PROGRAM MAIN
VAR
	traError			: BOOL;
	traInitDone			: BOOL;
	bModeOff			: BOOL;
	bModeManual			: BOOL := TRUE;
	bModeAuto			: BOOL;
	Err_T				: R_TRIG;
	Wrn_T				: R_TRIG;
	Wrn_T1				: R_TRIG;
	Reset_T				: R_TRIG;
	fbtimer				: TON;
	fbTimerSirens		: TON;
	fbTimer_IoT			: Ton;
	Run_T				: R_TRIG;
	Stop_T				: R_TRIG;
	k,k1				: INT;
	nState				: INT;
	nStateEmr			: INT;
	nState2				: INT;
	nState_IoT			: INT;
	bFaultFlag			: BOOL;
	nstateStop			: INT;
	fbTimerStop			: TON;
	timerStop			: ton;
	timerReset			: TON;
	nWriteData			: INT;
	TimerData			: TON;
	FbTimerModbus		: ARRAY [1..7] OF TON;
	fbEventlogger		: FB_Eventlogger;
	fbEventButton		: FB_EventButton;
	nstatechange		: INT;
	bWriteAlarm			: BOOL;
END_VAR

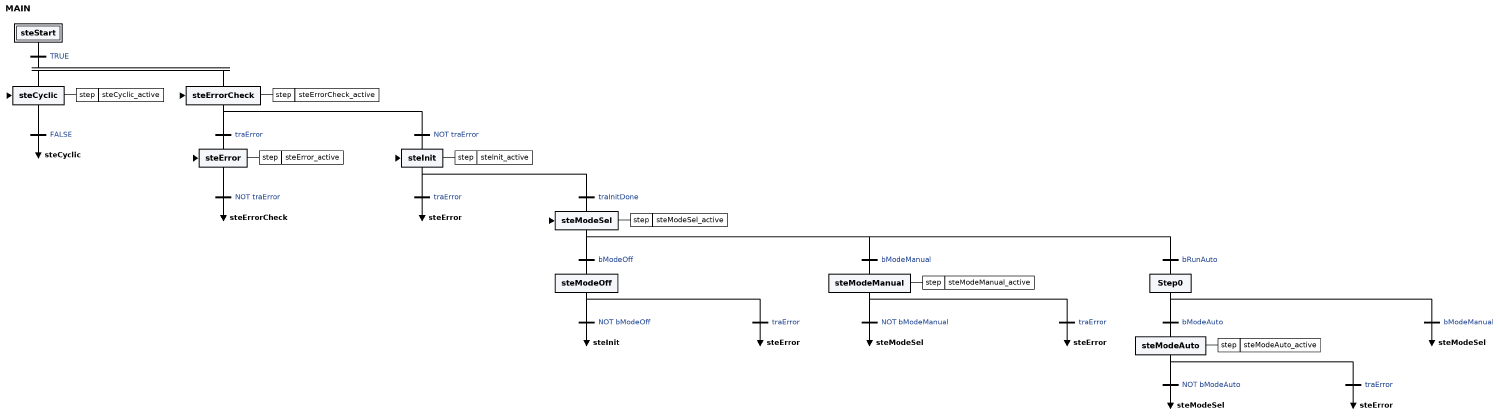
INITIAL_STEP steStart:
END_STEP
TRANSITION FROM steStart TO (steCyclic, steErrorCheck)
    := TRUE;
END_TRANSITION
STEP steCyclic:
    steCyclic_active(N);  // step action
END_STEP
TRANSITION FROM steCyclic TO steCyclic
    := FALSE;
END_TRANSITION
STEP steErrorCheck:
    steErrorCheck_active(N);  // step action
END_STEP
TRANSITION FROM steErrorCheck TO steError
    := traError;
END_TRANSITION
STEP steError:
    steError_active(N);  // step action
END_STEP
TRANSITION FROM steError TO steErrorCheck
    := NOT traError;
END_TRANSITION
TRANSITION FROM steErrorCheck TO steInit
    := NOT traError;
END_TRANSITION
STEP steInit:
    steInit_active(N);  // step action
END_STEP
TRANSITION FROM steInit TO steError
    := traError;
END_TRANSITION
TRANSITION FROM steInit TO steModeSel
    := traInitDone;
END_TRANSITION
STEP steModeSel:
    steModeSel_active(N);  // step action
END_STEP
TRANSITION FROM steModeSel TO steModeOff
    := bModeOff;
END_TRANSITION
STEP steModeOff:
END_STEP
TRANSITION FROM steModeOff TO steInit
    := NOT bModeOff;
END_TRANSITION
TRANSITION FROM steModeOff TO steError
    := traError;
END_TRANSITION
TRANSITION FROM steModeSel TO steModeManual
    := bModeManual;
END_TRANSITION
STEP steModeManual:
    steModeManual_active(N);  // step action
END_STEP
TRANSITION FROM steModeManual TO steModeSel
    := NOT bModeManual;
END_TRANSITION
TRANSITION FROM steModeManual TO steError
    := traError;
END_TRANSITION
TRANSITION FROM steModeSel TO Step0
    := bRunAuto;
END_TRANSITION
STEP Step0:
END_STEP
TRANSITION FROM Step0 TO steModeAuto
    := bModeAuto;
END_TRANSITION
TRANSITION FROM Step0 TO steModeSel
    := bModeManual;
END_TRANSITION
STEP steModeAuto:
    steModeAuto_active(N);  // step action
END_STEP
TRANSITION FROM steModeAuto TO steModeSel
    := NOT bModeAuto;
END_TRANSITION
TRANSITION FROM steModeAuto TO steError
    := traError;
END_TRANSITION

ACTION ListError:
Err_T(CLK := bError1);
Wrn_T(CLK := bWarning);

IF i > 100 THEN
	i := 100;
END_IF
		
CASE nState OF 
	0:
		IF Err_T.Q THEN
			nState := 1;
		ELSIF Wrn_T.Q THEN
			bWrn := TRUE;
			nState := 10;
		END_IF

	1:
		CASE nErrorID OF
			1:
				stErrorTxt := "E1_1.Lỗi hết hũ trạm 1 [kiểm tra U1I5-2]";
				stErrorTxt1 := 'E1_1.The jar is empty line 1 [check U1I5-2]';
				fbEventlogger(eventClass := TC_EVENTS.Entobel.Event1.uuidEventClass, nEventID := DINT_TO_UDINT(nErrorID));
			2:
				stErrorTxt := "E2_1.Lỗi hũ bị kẹt trạm 1 [kiểm tra U1I5-6]";
				stErrorTxt1 := 'E2_1.The jar  is trapped line 1 [check U1I5-6]';
				fbEventlogger(eventClass := TC_EVENTS.Entobel.Event2.uuidEventClass, nEventID := DINT_TO_UDINT(nErrorID));
			3:
				stErrorTxt := "E3_1.Lỗi ben chặn hũ trên rút về trạm 1 [kiểm tra U1I5-3]" ;
				stErrorTxt1 := 'E3_1.The upper cylinder retract  is faulty line 1 [check U1I5-3]';
				fbEventlogger(eventClass := TC_EVENTS.Entobel.Event3.uuidEventClass, nEventID := DINT_TO_UDINT(nErrorID));
			4:
				stErrorTxt := "E4_1.Lỗi ben chặn hũ dưới rút về trạm 1 [kiểm tra U1I5-4]";
				stErrorTxt1 := 'E4_1.The lower cylinder retract  is faulty line 1 [check U1I5-4]';
				fbEventlogger(eventClass := TC_EVENTS.Entobel.Event4.uuidEventClass, nEventID := DINT_TO_UDINT(nErrorID));
			5:
				stErrorTxt := "E5_1.Lỗi ben chặn hũ dưới đẩy ra trạm 1 [kiểmtra U1I5-5]";
				stErrorTxt1 := 'E5_1.The lower cylinder extend  is faulty line 1 [check U1I5-5]';
				fbEventlogger(eventClass := TC_EVENTS.Entobel.Event5.uuidEventClass, nEventID := DINT_TO_UDINT(nErrorID));
			6:
				stErrorTxt := "E6_1.Lỗi biến tần đảo thức ăn trạm 1 [kiểm tra biến tần 4]";
				stErrorTxt1 := 'E6_1.The inverter of agitator motor fault line 1 [check U1I5-6]';
				fbEventlogger(eventClass := TC_EVENTS.Entobel.Event6.uuidEventClass, nEventID := DINT_TO_UDINT(nErrorID));
			7:
				stErrorTxt := "E7_1.Lỗi driver chia thức ăn trạm 1 [kiểm tra driver 2]";
				stErrorTxt1 := 'E7_1.The driver of dispenser motor fault line 1 [check driver 2]';
				fbEventlogger(eventClass := TC_EVENTS.Entobel.Event7.uuidEventClass, nEventID := DINT_TO_UDINT(nErrorID));
			8:
				stErrorTxt := "E8_1.Lỗi ben chặn sâu rút về trạm 1 [kiểm tra U1I5-7]";
				stErrorTxt1 := 'E8_1.The cylinder blocking worm retract  is faulty line 1 [check U1I5-7]';
				fbEventlogger(eventClass := TC_EVENTS.Entobel.Event8.uuidEventClass, nEventID := DINT_TO_UDINT(nErrorID));
			9:
				stErrorTxt := "E9_1.Lỗi biến tần phểu rung sâu trạm 1 [kiểm tra biến tần 5]";
				stErrorTxt1 := 'E9_1.The inverter of vibrating funnel fault line 1 [check inverter 5]';
				fbEventlogger(eventClass := TC_EVENTS.Entobel.Event9.uuidEventClass, nEventID := DINT_TO_UDINT(nErrorID));
			10:
				stErrorTxt := "E10_1.Lỗi hết nắp trạm 1 [kiểm tra U1I5-8]";
				stErrorTxt1 := 'E10_1.The lid is empty line 1 [check U1I5-8]';
				fbEventlogger(eventClass := TC_EVENTS.Entobel.Event10.uuidEventClass, nEventID := DINT_TO_UDINT(nErrorID));
			11:
				stErrorTxt := "E11_1.Lỗi ben chặn nắp rút về trạm 1 [kiểm tra U1I6-1]";
				stErrorTxt1 := 'E11_1.The cylinder blocking the lid retract is faulty line 1 [check U1I6-1]';
				fbEventlogger(eventClass := TC_EVENTS.Entobel.Event11.uuidEventClass, nEventID := DINT_TO_UDINT(nErrorID));
			12:
				stErrorTxt := "E12-1.Lỗi ben chặn nắp đẩy ra trạm 1 [kiểm tra U1I6-2]";
				stErrorTxt1 := 'E12_1.The cylinder blocking the lid extend is faulty line 1 [check U1I6-2]';
				fbEventlogger(eventClass := TC_EVENTS.Entobel.Event12.uuidEventClass, nEventID := DINT_TO_UDINT(nErrorID));
			13:
				stErrorTxt := "E13_1.Lỗi ben hút/thả nắp rút về trạm 1 [kiểm tra U1I6-3]";
				stErrorTxt1 := 'E13_1.The cylinder sucking the lid retract is faulty line 1 [check U1I6-3]';
				fbEventlogger(eventClass := TC_EVENTS.Entobel.Event13.uuidEventClass, nEventID := DINT_TO_UDINT(nErrorID));
			14:
				stErrorTxt := "E14_1.Lỗi ben hút/thả nắp đẩy ra trạm 1 [kiểm tra U1I6-4]";
				stErrorTxt1 := 'E14_1.The cylinder sucking the lid extend is faulty line 1 [check U1I6-4]';
				fbEventlogger(eventClass := TC_EVENTS.Entobel.Event14.uuidEventClass, nEventID := DINT_TO_UDINT(nErrorID));
			15:
				stErrorTxt := "E15_1.Lỗi ben dập nắp rút về trạm 1 [kiểm tra U1I6-6]";
				stErrorTxt1 := 'E15_1.The cylinder pressing the lid retract is faulty line 1 [check U1I6-6]';
				fbEventlogger(eventClass := TC_EVENTS.Entobel.Event15.uuidEventClass, nEventID := DINT_TO_UDINT(nErrorID));
			16:
				stErrorTxt := "E16_1.Lỗi ben dập nắp đẩy ra trạm 1 [kiểm tra U1I6-7]";
				stErrorTxt1 := 'E16_1.The cylinder pressing the lid extend is faulty line 1 [check U1I6-7]';
				fbEventlogger(eventClass := TC_EVENTS.Entobel.Event16.uuidEventClass, nEventID := DINT_TO_UDINT(nErrorID));
			17:
				stErrorTxt := "E17_1.Lỗi ben lượt ra/vào rút về trạm 1 [kiểm tra U1I6-8]";
				stErrorTxt1 := 'E17_1.The comb cylinder retract is faulty line 1 [check U1I6-8]';
				fbEventlogger(eventClass := TC_EVENTS.Entobel.Event17.uuidEventClass, nEventID := DINT_TO_UDINT(nErrorID));
			18:
				stErrorTxt := "E18_1.Lỗi ben lượt ra/vào đẩy ra trạm 1 [kiểm tra U1I7-1]";
				stErrorTxt1 := 'E18_1.The comb cylinder extend is faulty line 1 [check U1I7-1]';
				fbEventlogger(eventClass := TC_EVENTS.Entobel.Event18.uuidEventClass, nEventID := DINT_TO_UDINT(nErrorID));
			19:
				stErrorTxt := "E19_1.Lỗi ben kẹp hũ rút về trạm 1 [kiểm tra U1I7-4]";
				stErrorTxt1 := 'E19_1.The clap cylinder retract is faulty line 1 [check U1I7-4]';
				fbEventlogger(eventClass := TC_EVENTS.Entobel.Event19.uuidEventClass, nEventID := DINT_TO_UDINT(nErrorID));
			20:
				stErrorTxt := "E20_1.Lỗi ben kẹp hũ đẩy ra trạm 1 [kiểm tra U1I7-5]";	
				stErrorTxt1 := 'E20_1.The clap cylinder extend is faulty line 1 [check U1I7-5]';
				fbEventlogger(eventClass := TC_EVENTS.Entobel.Event20.uuidEventClass, nEventID := DINT_TO_UDINT(nErrorID));
			21:
				stErrorTxt := "E21_1.Lỗi ben di chuyển lượt rút về trạm 1 [kiểm tra U1I7-2]";	
				stErrorTxt1 := 'E21_1.The cylinder moving comb retract is faulty line 1 [check U1I7-2]';
				fbEventlogger(eventClass := TC_EVENTS.Entobel.Event21.uuidEventClass, nEventID := DINT_TO_UDINT(nErrorID));
			22:
				stErrorTxt := "E22_1.Lỗi ben di chuyển lượt đẩy ra trạm 1 [kiểm tra U1I7-3]";
				stErrorTxt1 := 'E22_1.The cylinder moving comb extend is faulty line 1 [check U1I7-3]';
				fbEventlogger(eventClass := TC_EVENTS.Entobel.Event22.uuidEventClass, nEventID := DINT_TO_UDINT(nErrorID));
			45:
				stErrorTxt := "E23_1.Lỗi mất hũ khi đang cân thức ăn trạm 1 [kiểm tra U1I7-6]";
				stErrorTxt1 := 'E23_1.The jar is missed when weighting food line 1 [check U1I7-6]';
				fbEventlogger(eventClass := TC_EVENTS.Entobel.Event45.uuidEventClass, nEventID := DINT_TO_UDINT(nErrorID));
			47:
				stErrorTxt := "E24_1.Lỗi mất hũ khi đang cân sâu trạm 1 [kiểm tra U1I7-7]";
				stErrorTxt1 := 'E24_1.The jar is missed when weighting larvae line 1 [check U1I7-7]';
				fbEventlogger(eventClass := TC_EVENTS.Entobel.Event47.uuidEventClass, nEventID := DINT_TO_UDINT(nErrorID));
			49:
				stErrorTxt := "E25_1.Lỗi hút không được nắp trạm 1 [kiểm tra U1I6-5]";
				stErrorTxt1 := 'E25_1.Failed to suction the lid line 1 [check U1I6-5]';
				fbEventlogger(eventClass := TC_EVENTS.Entobel.Event49.uuidEventClass, nEventID := DINT_TO_UDINT(nErrorID));
			51:
				stErrorTxt := "E26_1.Lỗi nắp đã được hút trạm 1 [kiểm tra U1I6-5]";
				stErrorTxt1 := 'E26_1.The lid is still on the valve line 1 [check U1I5-6]';	
				fbEventlogger(eventClass := TC_EVENTS.Entobel.Event51.uuidEventClass, nEventID := DINT_TO_UDINT(nErrorID));
			53:
				stErrorTxt := "E27_1.Lỗi an toàn cửa 1 [kiểm tra U1I7-8]";	
				stErrorTxt1 := 'E27_1.The safety door 1 is error [check U1I7-8]';	
				fbEventlogger(eventClass := TC_EVENTS.Entobel.Event53.uuidEventClass, nEventID := DINT_TO_UDINT(nErrorID));
			54:
				stErrorTxt := "E28_1.Lỗi an toàn cửa 2 [kiểm tra U1I7-9]";
				stErrorTxt1 := 'E28_1.The safety door 2 is error [check U1I7-9]';	
				fbEventlogger(eventClass := TC_EVENTS.Entobel.Event54.uuidEventClass, nEventID := DINT_TO_UDINT(nErrorID));
			55:
				stErrorTxt := "E29_1.Lỗi an toàn cửa 3 [kiểm tra U1I7-10]";
				stErrorTxt1 := 'E29_1.The safety door 3 is error [check U1I7-10]';
				fbEventlogger(eventClass := TC_EVENTS.Entobel.Event55.uuidEventClass, nEventID := DINT_TO_UDINT(nErrorID));	
			56: 
				stErrorTxt := "E30_1.Lỗi quá cân thức ăn trạm 1 [kiểm tra cân thức ăn]";
				stErrorTxt1 := 'E30_1.Overload weightfood [check U1I5-6]';	
				fbEventlogger(eventClass := TC_EVENTS.Entobel.Event56.uuidEventClass, nEventID := DINT_TO_UDINT(nErrorID));
			57: 
				stErrorTxt := "E31_1.Lỗi quá cân sâu trạm 1 [kiểm tra cân sâu]";
				stErrorTxt1 := 'E30_1.Overload weightLarvae [check U1I5-6]';
				fbEventlogger(eventClass := TC_EVENTS.Entobel.Event57.uuidEventClass, nEventID := DINT_TO_UDINT(nErrorID));	
			60:
				stErrorTxt := "E32_1.Lỗi ben hút/thả hũ đẩy ra trạm 1 [kiểm tra U1I7-11]";
				stErrorTxt1 := 'E32_1.The cylinder sucking the jar is faulty line 1 [check U1I7-11]';
				fbEventlogger(eventClass := TC_EVENTS.Entobel.Event60.uuidEventClass, nEventID := DINT_TO_UDINT(nErrorID)); 
			64:
				stErrorTxt := "E33_1.Lỗi Modbus thiết bị 3";
				stErrorTxt1 := 'E33_1.Error Modbus device 3';
				fbEventlogger(eventClass := TC_EVENTS.Entobel.Event64.uuidEventClass, nEventID := DINT_TO_UDINT(nErrorID));	
			65:
				stErrorTxt := "E34_1.Lỗi Modbus thiết bị 4";
				stErrorTxt1 := 'E34_1.Error Modbus device 4';
				fbEventlogger(eventClass := TC_EVENTS.Entobel.Event65.uuidEventClass, nEventID := DINT_TO_UDINT(nErrorID));	
			66:
				stErrorTxt := "E35_1.Lỗi Modbus thiết bị 5";
				stErrorTxt1 := 'E35_1.Error Modbus device 5';
				fbEventlogger(eventClass := TC_EVENTS.Entobel.Event66.uuidEventClass, nEventID := DINT_TO_UDINT(nErrorID));	
			68:
				stErrorTxt := "E36_1.Lỗi Modbus thiết bị 7";
				stErrorTxt1 := 'E36_1.Error Modbus device 7';
				fbEventlogger(eventClass := TC_EVENTS.Entobel.Event68.uuidEventClass, nEventID := DINT_TO_UDINT(nErrorID));	
			69:
				stErrorTxt := "E37_1.Lỗi đầu cân thức ăn Mettler Toledo 1";
				stErrorTxt1 := 'E37_1.Error Mettler Toledo 1';
				fbEventlogger(eventClass := TC_EVENTS.Entobel.Event69.uuidEventClass, nEventID := DINT_TO_UDINT(nErrorID));	
			70:
				stErrorTxt := "E38_1.Lỗi đầu cân sâu Mettler Toledo 2";
				stErrorTxt1 := 'E38_1.Error Mettler Toledo 2';
				fbEventlogger(eventClass := TC_EVENTS.Entobel.Event70.uuidEventClass, nEventID := DINT_TO_UDINT(nErrorID));	
			73:
				stErrorTxt := "E39_1.Lỗi ben chặn sâu đẩy ra trạm 1 [kiểm tra U1I5-7]";
				stErrorTxt1 := 'E39_1.The cylinder blocking worm extend  is faulty line 1';
				fbEventlogger(eventClass := TC_EVENTS.Entobel.Event73.uuidEventClass, nEventID := DINT_TO_UDINT(nErrorID));	
			75:
				stErrorTxt := "E40_1.Lỗi thiếu khí đầu vào [kiểm tra U1I7-13]";
				stErrorTxt1 := 'E40_1.Error of lack of input air [check U1I7-13]';
				fbEventlogger(eventClass := TC_EVENTS.Entobel.Event75.uuidEventClass, nEventID := DINT_TO_UDINT(nErrorID));	
			76:
				stErrorTxt := "E41_1.Lỗi hết thức ăn trạm 1";
				stErrorTxt1 := 'E41_1.Error running out of food line 1';
				fbEventlogger(eventClass := TC_EVENTS.Entobel.Event76.uuidEventClass, nEventID := DINT_TO_UDINT(nErrorID));	
			77:
				stErrorTxt := "E42_1.Lỗi hết sâu trạm 1";
				stErrorTxt1 := 'E42_1.Error running out of larvae line 1';
				fbEventlogger(eventClass := TC_EVENTS.Entobel.Event78.uuidEventClass, nEventID := DINT_TO_UDINT(nErrorID));		
			98:
				stErrorTxt := "E98_1.Dừng khẩn [kiểm tra Emergency]";
				stErrorTxt1 := 'E98_1.Emergency Stop [check Emergency]';
				fbEventlogger(eventClass := TC_EVENTS.Entobel.Event98.uuidEventClass, nEventID := DINT_TO_UDINT(nErrorID));	 
			99: 
				stErrorTxt := "E99_1.Lỗi biến tần băng tải đầu ra [kiểm tra biến tần 3]";
				stErrorTxt1 := 'E99_1.The inverter of conveyor out [check inverter 3]';	
				fbEventlogger(eventClass := TC_EVENTS.Entobel.Event99.uuidEventClass, nEventID := DINT_TO_UDINT(nErrorID));
		END_CASE
		IF i <> 1 THEN
			FOR	k := i TO 2 BY -1 DO
				nErrorIDList1[k].nErrorID 	 := nErrorIDList1[k-1].nErrorID;
				nErrorIDList1[k].ErrorTime   := nErrorIDList1[k-1].ErrorTime;
				nErrorIDList1[k].ErrorStatus := nErrorIDList1[k-1].ErrorStatus;	
			END_FOR		
		END_IF 
		nErrorIDList1[1].nErrorID := nErrorID;
		nErrorIDList1[1].ErrorTime := SYSTEMTIME_TO_DT(GetLocalSystemTime.systemTime);
		nErrorIDList1[1].ErrorStatus := 1;
		nStatus1	:= 'ERROR';
		i := i + 1;
		bWarning := FALSE;
		bTo_alarm_side := TRUE;
		nState := 2;
	2:
		bWriteAlarm	:= TRUE;
		bSirens := TRUE;
		nState := 3;
	3:
		IF NOT bError1 THEN
			nState 	:= 0;
			bSirens := FALSE;
		END_IF
	10:
		CASE nWarningID OF
			101:
				stWarningTxt := "W1_1.Cảnh báo hết hũ trạm 1[kiểm tra U1I5-2]";
				stWarningTxt1 := 'W1_1.Warning out of jar line 1 [check U1I5-2]';
				fbEventlogger(eventClass := TC_EVENTS.Entobel.Event101.uuidEventClass, nEventID := DINT_TO_UDINT(nWarningID));
			102:
				stWarningTxt := "W2_1.Cảnh báo hết nắp trạm 1[kiểm tra U1I5-8]";
				stWarningTxt1 := 'W2_1.Warning out of lid line 1 [check U1I5-8]';
				fbEventlogger(eventClass := TC_EVENTS.Entobel.Event102.uuidEventClass, nEventID := DINT_TO_UDINT(nWarningID));
			103:
				stWarningTxt := "W3_1.Cảnh báo hết thức ăn trạm 1";
				stWarningTxt1 := 'W3_1.Warning running out of food line 1';
				fbEventlogger(eventClass := TC_EVENTS.Entobel.Event103.uuidEventClass, nEventID := DINT_TO_UDINT(nWarningID));
			104:
				stWarningTxt := "W4_1.Cảnh báo cân quá khối lượng thức ăn trạm 1";
				stWarningTxt1 := 'W4_1.Warning food weight exceeds limit line 1';
				fbEventlogger(eventClass := TC_EVENTS.Entobel.Event104.uuidEventClass, nEventID := DINT_TO_UDINT(nWarningID));
			105:
				stWarningTxt := "W5_1.Cảnh báo hết sâu trạm 1";
				stWarningTxt1 := 'W5_1.Warning running out of larvae line 1';
				fbEventlogger(eventClass := TC_EVENTS.Entobel.Event105.uuidEventClass, nEventID := DINT_TO_UDINT(nWarningID));
			106:
				stWarningTxt := "W6_1.Canh bao can qua khoi luong sau tram 1";
				stWarningTxt1 := 'W6_1.Warning larvae weight exceeds limit line 1';
				fbEventlogger(eventClass := TC_EVENTS.Entobel.Event106.uuidEventClass, nEventID := DINT_TO_UDINT(nWarningID));
			107:
				stWarningTxt := "W7_1.Cảnh báo dập nắp không vô trạm 1[kiểm tra U1I6-7]";
				stWarningTxt1 := 'W7_1.Warning do not press lid inward line 1 [check U1I6-7]';
				fbEventlogger(eventClass := TC_EVENTS.Entobel.Event107.uuidEventClass, nEventID := DINT_TO_UDINT(nWarningID));
			115:
				stWarningTxt := "W8_1.Cảnh báo mất kết nối với PC Advantech [kiểm tra PC]";
				stWarningTxt1 := 'W8_1.Warning disconnect to PC Advantech [check PC]';	
				bAlarm_Iot := TRUE;	
		END_CASE
		IF i <> 1 THEN
			FOR	k := i TO 2 BY -1 DO
				nErrorIDList1[k].nErrorID 	 := nErrorIDList1[k-1].nErrorID;
				nErrorIDList1[k].ErrorTime   := nErrorIDList1[k-1].ErrorTime;
				nErrorIDList1[k].ErrorStatus := nErrorIDList1[k-1].ErrorStatus;		
			END_FOR		
		END_IF 
		nErrorIDList1[1].nErrorID := nWarningID;
		nErrorIDList1[1].ErrorTime := SYSTEMTIME_TO_DT(GetLocalSystemTime.systemTime);
		nErrorIDList1[1].ErrorStatus := 1;
		nStatus1	:= 'WARNING';
		i := i + 1;
		nState := 11;
	11:
		bWriteAlarm	:= TRUE;
		bSirens := TRUE;
		nState := 12;
	12:
		bWarning := FALSE;
		nState := 0;		
END_CASE

IF bclearall THEN
	FOR k := 1 TO 100 DO
		AlarmList[1,k] := "";
		AlarmList[2,k] := "";	
		AlarmList[3,k] := "";
		AlarmList[4,k] := "";	
		AlarmList3[1,k] := '';
		AlarmList3[2,k] := '';	
		AlarmList3[3,k] := '';
		AlarmList3[4,k] := '';	
	END_FOR
	i := 1;
END_IF

IF username <> '' THEN
	IF getuser = 'Operator' THEN
		IF NOT bSafetyDoor1 THEN
			F_SetError(53,nLine := 3);
		ELSIF NOT bSafetyDoor2 THEN
			F_SetError(54,nLine := 3);	
		ELSIF NOT bSafetyDoor3 THEN
			F_SetError(55,nLine := 3);	
		END_IF
		bypass := FALSE;
		hienthibypass := FALSE;
	ELSIF getuser = 'Engineer' THEN
		hienthibypass := TRUE;
		IF NOT bypass THEN
			IF NOT bSafetyDoor1 THEN
				F_SetError(53,nLine := 3);
			ELSIF NOT bSafetyDoor2 THEN
				F_SetError(54,nLine := 3);	
			ELSIF NOT bSafetyDoor3 THEN
				F_SetError(55,nLine := 3);	
			END_IF
		END_IF
	END_IF
END_IF
IF username <> '' THEN
	IF Error[1] THEN 
		(*IF ErrorID[1] = 150 OR ErrorID[1] = 32 THEN
			FbTimerModbus[1](IN := FALSE, PT := T#1S);
		ELSE*)
			//FbTimerModbus[1](IN := TRUE, PT := T#1S);
			//IF FbTimerModbus[1].Q  THEN
				F_SetError(62,nLine := 2);
			//END_IF
		//END_IF
	ELSE
		FbTimerModbus[1](IN := FALSE);
	END_IF
	
	IF Error[2] THEN
		(*IF ErrorID[2] = 150 OR ErrorID[2] = 32 THEN
			FbTimerModbus[2](IN := FALSE, PT := T#1S);
		ELSE*)
			//FbTimerModbus[2](IN := TRUE, PT := T#1S);
			//IF FbTimerModbus[2].Q THEN
				F_SetError(63,nLine := 2);
			//END_IF
		//END_IF
	ELSE
		FbTimerModbus[2](IN := FALSE);
	END_IF
	
	IF Error[3] THEN
		(*IF ErrorID[3] = 150 OR ErrorID[3] = 32 THEN
			FbTimerModbus[3](IN := FALSE, PT := T#1S);
		ELSE*)
			//FbTimerModbus[3](IN := TRUE, PT := T#1S);
			//IF FbTimerModbus[3].Q THEN
				F_SetError(64,nLine := 3);
				PR_Conveyor_Out.Stop();
				bRun := FALSE;
			//END_IF
		//END_IF
	ELSE
		FbTimerModbus[3](IN := FALSE);
	END_IF
	
	IF Error[4] THEN
		(*IF ErrorID[4] = 150 OR ErrorID[4] = 32 THEN
			FbTimerModbus[4](IN := FALSE, PT := T#1S);
		ELSE *)
			//FbTimerModbus[4](IN := TRUE, PT := T#1S);
			//IF FbTimerModbus[4].Q THEN
				F_SetError(65,nLine := 1);
			//END_IF
		//END_IF
	ELSE
		FbTimerModbus[4](IN := FALSE);
	END_IF
	
	IF Error[5] THEN
		(*IF ErrorID[5] = 150 OR ErrorID[5] = 32 THEN
			FbTimerModbus[5](IN := FALSE, PT := T#1S);
		ELSE*)
			//FbTimerModbus[5](IN := TRUE, PT := T#1S);
			//IF FbTimerModbus[5].Q THEN
				F_SetError(66,nLine := 1);
			//END_IF
		//END_IF
	ELSE
		FbTimerModbus[5](IN := FALSE);
	END_IF
	
	IF Error[6] THEN
		(*IF ErrorID[6] = 150 OR ErrorID[6] = 32 THEN
			FbTimerModbus[6](IN := FALSE, PT := T#1S);
		ELSE*)
			//FbTimerModbus[6](IN := TRUE, PT := T#1S);
			//IF FbTimerModbus[6].Q THEN
				F_SetError(67,nLine := 2);
			//END_IF
		//END_IF
	ELSE
		FbTimerModbus[6](IN := FALSE);
	END_IF
	
	IF Error[7] THEN
		(*IF ErrorID[2] = 150 OR ErrorID[7] = 32 THEN
			FbTimerModbus[7](IN := FALSE, PT := T#1S);
		ELSE*)
			//FbTimerModbus[7](IN := TRUE, PT := T#1S);
			//IF FbTimerModbus[7].Q THEN
				F_SetError(68,nLine := 1);
			//END_IF
		//END_IF
	ELSE
		FbTimerModbus[7](IN := FALSE);
	END_IF
END_IF

IF username <> '' THEN
	IF bCheckVan THEN
		F_SetError(75,nLine := 3);
	END_IF
END_IF

IF bError1 AND bError2 AND (nErrorId = 99 OR nErrorID = 64) THEN
	PR_Conveyor_Out.Stop();
END_IF 

IF bWrn THEN
	bWrn2 := FALSE;
ELSIF bWrn2 THEN
	bWrn := FALSE;
END_IF

IF bWrn OR bWrn2 THEN
	bxoa := TRUE;
ELSE 
	bxoa := FALSE;
END_IF

CASE nStateEmr OF 
	0:
		IF NOT bEmer THEN
			F_SetError(98,nLine := 3);
			nStateEmr := 1;
		END_IF
	1:
		IF bEmer THEN
			nStateEmr := 0;
		END_IF
END_CASE
END_ACTION

ACTION MapRtig:
IF getuser = 'Operator' THEN
	CASE nstatechange OF 
		0:
			//line 1
			fFast_Speed_line1_change						:= PR_Line01.fFast_Speed;//FoodWeight
			fSlow_Speed_1_line1_change						:= PR_Line01.fSlow_Speed_1;
			fSlow_Speed_2_line1_change						:= PR_Line01.fSlow_Speed_2;
			fDerisedWeight_Food_line1_change				:= PR_Line01.fDerisedWeight_Food;
			fChangeMode_Food_1_line1_change					:= PR_Line01.fChangeMode_Food_1;
			fChangeMode_Food_2_line1_change					:= PR_Line01.fChangeMode_Food_2;
			fPerStop_Food_line1_change						:= PR_Line01.fPerStop_Food;
			fTimer_Check_Food_line1_change					:= PR_Line01.fTimer_Check_Food;
			fDelta_Food_line1_change						:= PR_Line01.fDelta_Food;
			fFast_Speed_vibrating_funnel_line1_change		:= PR_Line01.fFast_Speed_vibrating_funnel;//WormWeight
			fSlow_Speed_vibrating_funnel_1_line1_change		:= PR_Line01.fSlow_Speed_vibrating_funnel_1;
			fSlow_Speed_vibrating_funnel_2_line1_change		:= PR_Line01.fSlow_Speed_vibrating_funnel_2;
			fDerisedWeight_Worm_line1_change				:= PR_Line01.fDerisedWeight_Worm;
			fChangeMode_Worm_1_line1_change					:= PR_Line01.fChangeMode_Worm_1;
			fChangeMode_Worm_2_line1_change					:= PR_Line01.fChangeMode_Worm_2;
			fPerStop_Worm_line1_change						:= PR_Line01.fPerStop_Worm;
			fTimer_Check_Worm_line1_change					:= PR_Line01.fTimer_Check_Worm;
			fDelta_Worm_line1_change						:= PR_Line01.fDelta_Worm;
			//line 2
			fFast_Speed_line2_change						:= PR_Line02.fFast_Speed;//FoodWeight
			fSlow_Speed_1_line2_change						:= PR_Line02.fSlow_Speed_1;
			fSlow_Speed_2_line2_change						:= PR_Line02.fSlow_Speed_2;
			fDerisedWeight_Food_line2_change				:= PR_Line02.fDerisedWeight_Food;
			fChangeMode_Food_1_line2_change					:= PR_Line02.fChangeMode_Food_1;
			fChangeMode_Food_2_line2_change					:= PR_Line02.fChangeMode_Food_2;
			fPerStop_Food_line2_change						:= PR_Line02.fPerStop_Food;
			fTimer_Check_Food_line2_change					:= PR_Line02.fTimer_Check_Food;
			fDelta_Food_line2_change						:= PR_Line02.fDelta_Food;
			fFast_Speed_vibrating_funnel_line2_change		:= PR_Line02.fFast_Speed_vibrating_funnel;//WormWeight
			fSlow_Speed_vibrating_funnel_1_line2_change		:= PR_Line02.fSlow_Speed_vibrating_funnel_1;
			fSlow_Speed_vibrating_funnel_2_line2_change		:= PR_Line02.fSlow_Speed_vibrating_funnel_2;
			fDerisedWeight_Worm_line2_change				:= PR_Line02.fDerisedWeight_Worm;
			fChangeMode_Worm_1_line2_change					:= PR_Line02.fChangeMode_Worm_1;
			fChangeMode_Worm_2_line2_change					:= PR_Line02.fChangeMode_Worm_2;
			fPerStop_Worm_line2_change						:= PR_Line02.fPerStop_Worm;
			fTimer_Check_Worm_line2_change					:= PR_Line02.fTimer_Check_Worm;
			fDelta_Worm_line2_change						:= PR_Line02.fDelta_Worm;
			nstatechange := 1;
		1:
			IF 	fFast_Speed_line1_change <> PR_Line01.fFast_Speed THEN
				fbEventButton(eventClass := TC_EVENTS.Entobel.Event150.uuidEventClass, nEventID := 150,
							  sString := REAL_TO_STRING(PR_Line01.fFast_Speed));
				nstatechange := 0;
			ELSIF fSlow_Speed_1_line1_change <> PR_Line01.fSlow_Speed_1 THEN
				fbEventButton(eventClass := TC_EVENTS.Entobel.Event151.uuidEventClass, nEventID := 151,
							  sString := REAL_TO_STRING(PR_Line01.fSlow_Speed_1)); 
				nstatechange := 0;
			ELSIF fSlow_Speed_2_line1_change <> PR_Line01.fSlow_Speed_2 THEN
				fbEventButton(eventClass := TC_EVENTS.Entobel.Event152.uuidEventClass, nEventID := 152,
							  sString := REAL_TO_STRING(PR_Line01.fSlow_Speed_2)); 
				nstatechange := 0;
			ELSIF fDerisedWeight_Food_line1_change <> PR_Line01.fDerisedWeight_Food THEN
				fbEventButton(eventClass := TC_EVENTS.Entobel.Event153.uuidEventClass, nEventID := 153,
							  sString := REAL_TO_STRING(PR_Line01.fDerisedWeight_Food)); 
				nstatechange := 0;
			ELSIF fChangeMode_Food_1_line1_change <> PR_Line01.fChangeMode_Food_1 THEN
				fbEventButton(eventClass := TC_EVENTS.Entobel.Event154.uuidEventClass, nEventID := 154,
							  sString := REAL_TO_STRING(PR_Line01.fChangeMode_Food_1)); 
				nstatechange := 0;
			ELSIF fChangeMode_Food_2_line1_change <> PR_Line01.fChangeMode_Food_2 THEN
				fbEventButton(eventClass := TC_EVENTS.Entobel.Event155.uuidEventClass, nEventID := 155,
							  sString := REAL_TO_STRING(PR_Line01.fChangeMode_Food_2)); 
				nstatechange := 0;
			ELSIF fPerStop_Food_line1_change <> PR_Line01.fPerStop_Food THEN
				fbEventButton(eventClass := TC_EVENTS.Entobel.Event156.uuidEventClass, nEventID := 156,
							  sString := REAL_TO_STRING(PR_Line01.fPerStop_Food)); 
				nstatechange := 0;
			ELSIF fTimer_Check_Food_line1_change <> PR_Line01.fTimer_Check_Food THEN
				fbEventButton(eventClass := TC_EVENTS.Entobel.Event157.uuidEventClass, nEventID := 157,
							  sString := REAL_TO_STRING(PR_Line01.fTimer_Check_Food)); 
				nstatechange := 0;
			ELSIF fDelta_Food_line1_change <> PR_Line01.fDelta_Food THEN
				fbEventButton(eventClass := TC_EVENTS.Entobel.Event158.uuidEventClass, nEventID := 158,
							  sString := REAL_TO_STRING(PR_Line01.fDelta_Food)); 
				nstatechange := 0;
			ELSIF fFast_Speed_vibrating_funnel_line1_change <> PR_Line01.fFast_Speed_vibrating_funnel THEN
					fbEventButton(eventClass := TC_EVENTS.Entobel.Event159.uuidEventClass, nEventID := 159,
							  sString := REAL_TO_STRING(PR_Line01.fFast_Speed_vibrating_funnel)); 
				nstatechange := 0;
			ELSIF fSlow_Speed_vibrating_funnel_1_line1_change <> PR_Line01.fSlow_Speed_vibrating_funnel_1 THEN
				fbEventButton(eventClass := TC_EVENTS.Entobel.Event160.uuidEventClass, nEventID := 160,
							  sString := REAL_TO_STRING(PR_Line01.fSlow_Speed_vibrating_funnel_1)); 
				nstatechange := 0;
			ELSIF fSlow_Speed_vibrating_funnel_2_line1_change <> PR_Line01.fSlow_Speed_vibrating_funnel_2 THEN
				fbEventButton(eventClass := TC_EVENTS.Entobel.Event161.uuidEventClass, nEventID := 161,
							  sString := REAL_TO_STRING(PR_Line01.fSlow_Speed_vibrating_funnel_2)); 
				nstatechange := 0;
			ELSIF fDerisedWeight_Worm_line1_change <> PR_Line01.fDerisedWeight_Worm THEN
				fbEventButton(eventClass := TC_EVENTS.Entobel.Event162.uuidEventClass, nEventID := 162,
							  sString := REAL_TO_STRING(PR_Line01.fDerisedWeight_Worm)); 
				nstatechange := 0;
			ELSIF fChangeMode_Worm_1_line1_change <> PR_Line01.fChangeMode_Worm_1 THEN
				fbEventButton(eventClass := TC_EVENTS.Entobel.Event163.uuidEventClass, nEventID := 163,
							  sString := REAL_TO_STRING(PR_Line01.fChangeMode_Worm_1)); 
				nstatechange := 0;
			ELSIF fChangeMode_Worm_2_line1_change <> PR_Line01.fChangeMode_Worm_2 THEN
				fbEventButton(eventClass := TC_EVENTS.Entobel.Event164.uuidEventClass, nEventID := 164,
							  sString := REAL_TO_STRING(PR_Line01.fChangeMode_Worm_2)); 
				nstatechange := 0;
			ELSIF fPerStop_Worm_line1_change <> PR_Line01.fPerStop_Worm THEN
				fbEventButton(eventClass := TC_EVENTS.Entobel.Event165.uuidEventClass, nEventID := 165,
							  sString := REAL_TO_STRING(PR_Line01.fPerStop_Worm)); 
				nstatechange := 0;
			ELSIF fTimer_Check_Worm_line1_change <> PR_Line01.fTimer_Check_Worm THEN
				fbEventButton(eventClass := TC_EVENTS.Entobel.Event166.uuidEventClass, nEventID := 166,
							  sString := REAL_TO_STRING(PR_Line01.fTimer_Check_Worm)); 
				nstatechange := 0;
			ELSIF fDelta_Worm_line1_change <> PR_Line01.fDelta_Worm THEN
				fbEventButton(eventClass := TC_EVENTS.Entobel.Event167.uuidEventClass, nEventID := 167,
							  sString := REAL_TO_STRING(PR_Line01.fDelta_Worm)); 
				nstatechange := 0;
			ELSIF 	fFast_Speed_line2_change <> PR_Line02.fFast_Speed THEN
				fbEventButton(eventClass := TC_EVENTS.Entobel.Event168.uuidEventClass, nEventID := 168,
							  sString := REAL_TO_STRING(PR_Line02.fFast_Speed));
				nstatechange := 0;
			ELSIF fSlow_Speed_1_line2_change <> PR_Line02.fSlow_Speed_1 THEN
				fbEventButton(eventClass := TC_EVENTS.Entobel.Event169.uuidEventClass, nEventID := 169,
							  sString := REAL_TO_STRING(PR_Line02.fSlow_Speed_1)); 
				nstatechange := 0;
			ELSIF fSlow_Speed_2_line2_change <> PR_Line02.fSlow_Speed_2 THEN
				fbEventButton(eventClass := TC_EVENTS.Entobel.Event170.uuidEventClass, nEventID := 170,
							  sString := REAL_TO_STRING(PR_Line02.fSlow_Speed_2)); 
				nstatechange := 0;
			ELSIF fDerisedWeight_Food_line2_change <> PR_Line02.fDerisedWeight_Food THEN
				fbEventButton(eventClass := TC_EVENTS.Entobel.Event171.uuidEventClass, nEventID := 171,
							  sString := REAL_TO_STRING(PR_Line02.fDerisedWeight_Food)); 
				nstatechange := 0;
			ELSIF fChangeMode_Food_1_line2_change <> PR_Line02.fChangeMode_Food_1 THEN
				fbEventButton(eventClass := TC_EVENTS.Entobel.Event172.uuidEventClass, nEventID := 172,
							  sString := REAL_TO_STRING(PR_Line02.fChangeMode_Food_1)); 
				nstatechange := 0;
			ELSIF fChangeMode_Food_2_line2_change <> PR_Line02.fChangeMode_Food_2 THEN
				fbEventButton(eventClass := TC_EVENTS.Entobel.Event173.uuidEventClass, nEventID := 173,
							  sString := REAL_TO_STRING(PR_Line02.fChangeMode_Food_2)); 
				nstatechange := 0;
			ELSIF fPerStop_Food_line2_change <> PR_Line02.fPerStop_Food THEN
				fbEventButton(eventClass := TC_EVENTS.Entobel.Event174.uuidEventClass, nEventID := 174,
							  sString := REAL_TO_STRING(PR_Line02.fPerStop_Food)); 
				nstatechange := 0;
			ELSIF fTimer_Check_Food_line2_change <> PR_Line02.fTimer_Check_Food THEN
				fbEventButton(eventClass := TC_EVENTS.Entobel.Event175.uuidEventClass, nEventID := 175,
							  sString := REAL_TO_STRING(PR_Line02.fTimer_Check_Food)); 
				nstatechange := 0;
			ELSIF fDelta_Food_line2_change <> PR_Line02.fDelta_Food THEN
				fbEventButton(eventClass := TC_EVENTS.Entobel.Event176.uuidEventClass, nEventID := 176,
							  sString := REAL_TO_STRING(PR_Line02.fDelta_Food)); 
				nstatechange := 0;
			ELSIF fFast_Speed_vibrating_funnel_line2_change <> PR_Line02.fFast_Speed_vibrating_funnel THEN
				fbEventButton(eventClass := TC_EVENTS.Entobel.Event185.uuidEventClass, nEventID := 185,
							  sString := REAL_TO_STRING(PR_Line02.fFast_Speed_vibrating_funnel)); 
				nstatechange := 0;
			ELSIF fSlow_Speed_vibrating_funnel_1_line2_change <> PR_Line02.fSlow_Speed_vibrating_funnel_1 THEN
				fbEventButton(eventClass := TC_EVENTS.Entobel.Event177.uuidEventClass, nEventID := 177,
							  sString := REAL_TO_STRING(PR_Line02.fSlow_Speed_vibrating_funnel_1)); 
				nstatechange := 0;
			ELSIF fSlow_Speed_vibrating_funnel_2_line2_change <> PR_Line02.fSlow_Speed_vibrating_funnel_2 THEN
				fbEventButton(eventClass := TC_EVENTS.Entobel.Event178.uuidEventClass, nEventID := 178,
							  sString := REAL_TO_STRING(PR_Line02.fSlow_Speed_vibrating_funnel_2)); 
				nstatechange := 0;
			ELSIF fDerisedWeight_Worm_line2_change <> PR_Line02.fDerisedWeight_Worm THEN
				fbEventButton(eventClass := TC_EVENTS.Entobel.Event179.uuidEventClass, nEventID := 179,
							  sString := REAL_TO_STRING(PR_Line02.fDerisedWeight_Worm)); 
				nstatechange := 0;
			ELSIF fChangeMode_Worm_1_line2_change <> PR_Line02.fChangeMode_Worm_1 THEN
				fbEventButton(eventClass := TC_EVENTS.Entobel.Event180.uuidEventClass, nEventID := 180,
							  sString := REAL_TO_STRING(PR_Line02.fChangeMode_Worm_1)); 
				nstatechange := 0;
			ELSIF fChangeMode_Worm_2_line2_change <> PR_Line02.fChangeMode_Worm_2 THEN
				fbEventButton(eventClass := TC_EVENTS.Entobel.Event181.uuidEventClass, nEventID := 181,
							  sString := REAL_TO_STRING(PR_Line02.fChangeMode_Worm_2)); 
				nstatechange := 0;
			ELSIF fPerStop_Worm_line2_change <> PR_Line02.fPerStop_Worm THEN
				fbEventButton(eventClass := TC_EVENTS.Entobel.Event182.uuidEventClass, nEventID := 182,
							  sString := REAL_TO_STRING(PR_Line02.fPerStop_Worm)); 
				nstatechange := 0;
			ELSIF fTimer_Check_Worm_line2_change <> PR_Line02.fTimer_Check_Worm THEN
				fbEventButton(eventClass := TC_EVENTS.Entobel.Event183.uuidEventClass, nEventID := 183,
							  sString := REAL_TO_STRING(PR_Line02.fTimer_Check_Worm)); 
				nstatechange := 0;
			ELSIF fDelta_Worm_line2_change <> PR_Line02.fDelta_Worm THEN
				fbEventButton(eventClass := TC_EVENTS.Entobel.Event184.uuidEventClass, nEventID := 184,
							  sString := REAL_TO_STRING(PR_Line02.fDelta_Worm)); 
				nstatechange := 0;
			END_IF
	END_CASE
END_IF
END_ACTION

ACTION Reset_active:
PR_Line01.Reset();
END_ACTION

ACTION Start_active:
PR_Conveyor_Out.Stop();
END_ACTION

ACTION steCyclic_active:
PR_Line01();
PR_Conveyor_Out();
MapRtig();
ListError();
PRG_MainRecipe1();
GetLocalSystemTime(bEnable := 1,);
SystemTimeFull 	:= SYSTEMTIME_TO_STRING(in := GetLocalSystemTime.systemTime);
Onlyday 	:= MID(STR:= SystemTimeFull, LEN:=10 , POS:=1 );
OnlyTime 	:= MID(STR:= SystemTimeFull, LEN:=8 , POS:=12 );
//login
IF username <> '' THEN
	openstartpage := TRUE;
ELSE
	openstartpage := FALSE;
END_IF
getuser := WSTRING_TO_STRING(VisuElems.CurrentUserGroupName);

IF VisuElems.CURRENTLANGUAGE = 'vn' THEN
	GVL_OF_VU.bVN := TRUE;
ELSE
	GVL_OF_VU.bVN := FALSE;
END_IF

IF NOT bEmer THEN
	PR_Conveyor_Out.Stop();
	traError := TRUE;
	bLight_Running := FALSE;
	bLight_Stop := TRUE;
END_IF

IF bError1 THEN 
	traError := TRUE;
END_IF

Run_conveyor(CLK := bStart);
Stop_conveyor(CLK := bStop);
IF Run_conveyor.Q THEN
	status := 'RUN';
	bRun := TRUE;
	bStopConv := FALSE;
END_IF

IF bReset THEN
	bWarning := FALSE;
END_IF

IF Stop_conveyor.Q THEN
	bStopConv := TRUE;
	bRun := FALSE;
END_IF

IF bStart THEN
	bfinish1 := TRUE;
	bfinish2 := TRUE;
END_IF

IF bRun THEN
	PR_Conveyor_Out.Auto();
	bLight_Running := TRUE;
	bLight_Stop	:= FALSE;
ELSIF bStopConv AND bfinish1 AND bfinish2 THEN
	PR_Conveyor_Out.Stop();
	status := 'STOP';
	bRun := FALSE;
	bLight_Running := FALSE;
	bLight_Stop	:= TRUE;
END_IF

CASE nWriteData OF 
	0:
		TimerData(IN := TRUE, PT := T#0.5S);
		WritePSData(NETID:='', PORT:=851, START:=FALSE, TMOUT:=T#1S );
		IF TimerData.Q THEN
			nWriteData := 1;
		END_IF
	1:
		TimerData(IN := FALSE);
		nWriteData := 2;
	2:
		TimerData(IN := TRUE, PT := T#0.5S);
		WritePSData(NETID:='', PORT:=851, START:= TRUE, TMOUT:=T#1S );
		IF TimerData.Q THEN
			nWriteData := 3;
		END_IF
	3:
		TimerData(IN := FALSE);
		nWriteData := 0;
END_CASE

IF PR_Conveyor_Out.fb_Conveyor.fbInverter.bVFD THEN
	bRunAuto := TRUE;
ELSE
	bRunAuto := false;
END_IF

CASE nState_IoT OF
	0:
		IF bAlarm THEN
			nState_IoT := 1;
		ELSE
			fbTimer_IoT(IN := TRUE, PT := T#10S);
			IF fbTimer_IoT.Q THEN
				F_SetWarning(115,1);
				F_SetWarning(115,2);
				nState_IoT := 2;
			END_IF
		END_IF
	1:
		bAlarm := FALSE;
		fbTimer_IoT(IN := FALSE);
		nState_IoT := 0;
	2:
		fbTimer_IoT(IN := FALSE);
		IF bAlarm OR bReset THEN
			bWrn := FALSE;
			bWrn2 := FALSE;
			bAlarm_Iot := FALSE;
			nState_IoT := 0;
			bSirens := FALSE;
		END_IF
END_CASE
//Error List
IF bWriteAlarm THEN
FOR k1 := 1 TO 100 DO
	AlarmList[1,k1] 	:= INT_TO_WSTRING(nErrorIDList1[k1].nErrorID);
	AlarmList3[1,k1]	:= INT_TO_STRING(nErrorIDList1[k1].nErrorID);
	AlarmList[4,k1] 	:= STRING_TO_WSTRING(MID(STR := DT_TO_STRING(nErrorIDList1[k1].ErrorTime),LEN := 19, POS := 4));
	AlarmList3[4,k1] 	:= MID(STR := DT_TO_STRING(nErrorIDList1[k1].ErrorTime),LEN := 19, POS := 4);
	IF nErrorIDList1[k1].ErrorStatus = 1 THEN
		AlarmList[3,k1] := "Active";
		AlarmList3[3,k1] := 'Active';
	ELSE
		AlarmList[3,k1] := "Release";
		AlarmList3[3,k1] := 'Release';
	END_IF
	CASE nErrorIDList1[k1].nErrorID OF
			0: 
				AlarmList[4,k1] := "";
				AlarmList[3,k1] := "";
				AlarmList3[4,k1] := '';
				AlarmList3[3,k1] := '';
			1:
				AlarmList[2,k1]  := "E1_1.Lỗi hết hũ trạm 1 [kiểm tra U1I5-2]";
				AlarmList3[2,k1] := 'E1_1.The jar is empty line 1 [check U1I5-2]';
			2:
				AlarmList[2,k1] := "E2_1.Lỗi hũ bị kẹt trạm 1 [kiểm tra U1I5-6]";
				AlarmList3[2,k1] := 'E2_1.The jar  is trapped line 1 [check U1I5-6]';
			3:
				AlarmList[2,k1] := "E3_1.Lỗi ben chặn hũ trên rút về trạm 1 [kiểm tra U1I5-3]" ;
				AlarmList3[2,k1] := 'E3_1.The upper cylinder retract  is faulty line 1 [check U1I5-3]';
			4:
				AlarmList[2,k1] := "E4_1.Lỗi ben chặn hũ dưới rút về trạm 1 [kiểm tra U1I5-4]";
				AlarmList3[2,k1] := 'E4_1.The lower cylinder retract  is faulty line 1 [check U1I5-4]';
			5:
				AlarmList[2,k1] := "E5_1.Lỗi ben chặn hũ dưới đẩy ra trạm 1 [kiểmtra U1I5-5]";
				AlarmList3[2,k1] := 'E5_1.The lower cylinder extend  is faulty line 1 [check U1I5-5]';
			6:
				AlarmList[2,k1] := "E6_1.Lỗi biến tần đảo thức ăn trạm 1 [kiểm tra biến tần 4]";
				AlarmList3[2,k1] := 'E6_1.The inverter of agitator motor fault line 1 [check U1I5-6]';
			7:
				AlarmList[2,k1] := "E7_1.Lỗi driver chia thức ăn trạm 1 [kiểm tra driver 2]";
				AlarmList3[2,k1] := 'E7_1.The driver of dispenser motor fault line 1 [check driver 2]';
			8:
				AlarmList[2,k1] := "E8_1.Lỗi ben chặn sâu rút về trạm 1 [kiểm tra U1I5-7]";
				AlarmList3[2,k1] := 'E8_1.The cylinder blocking worm retract  is faulty line 1 [check U1I5-7]';
			9:
				AlarmList[2,k1] := "E9_1.Lỗi biến tần phểu rung sâu trạm 1 [kiểm tra biến tần 5]";
				AlarmList3[2,k1] := 'E9_1.The inverter of vibrating funnel fault line 1 [check inverter 5]';
			10:
				AlarmList[2,k1] := "E10_1.Lỗi hết nắp trạm 1 [kiểm tra U1I5-8]";
				AlarmList3[2,k1] := 'E10_1.The lid is empty line 1 [check U1I5-8]';
			11:
				AlarmList[2,k1] := "E11_1.Lỗi ben chặn nắp rút về trạm 1 [kiểm tra U1I6-1]";
				AlarmList3[2,k1] := 'E11_1.The cylinder blocking the lid retract is faulty line 1 [check U1I6-1]';
			12:
				AlarmList[2,k1] := "E12-1.Lỗi ben chặn nắp đẩy ra trạm 1 [kiểm tra U1I6-2]";
				AlarmList3[2,k1] := 'E12_1.The cylinder blocking the lid extend is faulty line 1 [check U1I6-2]';
			13:
				AlarmList[2,k1] := "E13_1.Lỗi ben hút/thả nắp rút về trạm 1 [kiểm tra U1I6-3]";
				AlarmList3[2,k1] := 'E13_1.The cylinder sucking the lid retract is faulty line 1 [check U1I6-3]';
			14:
				AlarmList[2,k1] := "E14_1.Lỗi ben hút/thả nắp đẩy ra trạm 1 [kiểm tra U1I6-4]";
				AlarmList3[2,k1] := 'E14_1.The cylinder sucking the lid extend is faulty line 1 [check U1I6-4]';
			15:
				AlarmList[2,k1] := "E15_1.Lỗi ben dập nắp rút về trạm 1 [kiểm tra U1I6-6]";
				AlarmList3[2,k1] := 'E15_1.The cylinder pressing the lid retract is faulty line 1 [check U1I6-6]';
			16:
				AlarmList[2,k1] := "E16_1.Lỗi ben dập nắp đẩy ra trạm 1 [kiểm tra U1I6-7]";
				AlarmList3[2,k1] := 'E16_1.The cylinder pressing the lid extend is faulty line 1 [check U1I6-7]';
			17:
				AlarmList[2,k1] := "E17_1.Lỗi ben lượt ra/vào rút về trạm 1 [kiểm tra U1I6-8]";
				AlarmList3[2,k1] := 'E17_1.The comb cylinder retract is faulty line 1 [check U1I6-8]';
			18:
				AlarmList[2,k1] := "E18_1.Lỗi ben lượt ra/vào đẩy ra trạm 1 [kiểm tra U1I7-1]";
				AlarmList3[2,k1] := 'E18_1.The comb cylinder extend is faulty line 1 [check U1I7-1]';
			19:
				AlarmList[2,k1] := "E19_1.Lỗi ben kẹp hũ rút về trạm 1 [kiểm tra U1I7-4]";
				AlarmList3[2,k1] := 'E19_1.The clap cylinder retract is faulty line 1 [check U1I7-4]';
			20:
				AlarmList[2,k1] := "E20_1.Lỗi ben kẹp hũ đẩy ra trạm 1 [kiểm tra U1I7-5]";	
				AlarmList3[2,k1] := 'E20_1.The clap cylinder extend is faulty line 1 [check U1I7-5]';
			21:
				AlarmList[2,k1] := "E21_1.Lỗi ben di chuyển lượt rút về trạm 1 [kiểm tra U1I7-2]";	
				AlarmList3[2,k1] := 'E21_1.The cylinder moving comb retract is faulty line 1 [check U1I7-2]';
			22:
				AlarmList[2,k1] := "E22_1.Lỗi ben di chuyển lượt đẩy ra trạm 1 [kiểm tra U1I7-3]";
				AlarmList3[2,k1] := 'E22_1.The cylinder moving comb extend is faulty line 1 [check U1I7-3]';
			45:
				AlarmList[2,k1] := "E23_1.Lỗi mất hũ khi đang cân thức ăn trạm 1 [kiểm tra U1I7-6]";
				AlarmList3[2,k1] := 'E23_1.The jar is missed when weighting food line 1 [check U1I7-6]';
			47:
				AlarmList[2,k1] := "E24_1.Lỗi mất hũ khi đang cân sâu trạm 1 [kiểm tra U1I7-7]";
				AlarmList3[2,k1] := 'E24_1.The jar is missed when weighting larvae line 1 [check U1I7-7]';
			49:
				AlarmList[2,k1] := "E25_1.Lỗi hút không được nắp trạm 1 [kiểm tra U1I6-5]";
				AlarmList3[2,k1] := 'E25_1.Failed to suction the lid line 1 [check U1I6-5]';
			51:
				AlarmList[2,k1] := "E26_1.Lỗi nắp đã được hút trạm 1 [kiểm tra U1I6-5]";
				AlarmList3[2,k1] := 'E26_1.The lid is still on the valve line 1 [check U1I5-6]';
			53:
				AlarmList[2,k1] := "E27_1.Lỗi an toàn cửa 1 [kiểm tra U1I7-8]";	
				AlarmList3[2,k1] := 'E27_1.The safety door 1 is error [check U1I7-8]';
			54:
				AlarmList[2,k1] := "E28_1.Lỗi an toàn cửa 2 [kiểm tra U1I7-9]";
				AlarmList3[2,k1] := 'E28_1.The safety door 2 is error [check U1I7-9]';
			55:
				AlarmList[2,k1] := "E29_1.Lỗi an toàn cửa 3 [kiểm tra U1I7-10]";
				AlarmList3[2,k1] := 'E29_1.The safety door 3 is error [check U1I7-10]';
			56: 
				AlarmList[2,k1] := "E30_1.Lỗi quá cân thức ăn trạm 1 [kiểm tra cân thức ăn]";
				AlarmList3[2,k1] := 'E30_1.Overload weightfood [check U1I5-6]';
			57: 
				AlarmList[2,k1] := "E31_1.Lỗi quá cân sâu trạm 1 [kiểm tra cân sâu]";
				AlarmList3[2,k1] := 'E30_1.Overload weightLarvae [check U1I5-6]';	
			60:
				AlarmList[2,k1] := "E32_1.Lỗi ben hút/thả hũ đẩy ra trạm 1 [kiểm tra U1I7-11]";
				AlarmList3[2,k1] := 'E32_1.The cylinder sucking the jar is faulty line 1 [check U1I7-11]'; 
			64:
				AlarmList[2,k1] := "E33_1.Lỗi Modbus thiết bị 3";
				AlarmList3[2,k1] := 'E33_1.Error Modbus device 3';	
			65:
				AlarmList[2,k1] := "E34_1.Lỗi Modbus thiết bị 4";
				AlarmList3[2,k1] := 'E34_1.Error Modbus device 4';
			66:
				AlarmList[2,k1] := "E35_1.Lỗi Modbus thiết bị 5";
				AlarmList3[2,k1] := 'E35_1.Error Modbus device 5';	
			68:
				AlarmList[2,k1] := "E36_1.Lỗi Modbus thiết bị 7";
				AlarmList3[2,k1] := 'E36_1.Error Modbus device 7';	
			69:
				AlarmList[2,k1] := "E37_1.Lỗi đầu cân thức ăn Mettler Toledo 1";
				AlarmList3[2,k1] := 'E37_1.Error Mettler Toledo 1';	
			70:
				AlarmList[2,k1] := "E38_1.Lỗi đầu cân sâu Mettler Toledo 2";
				AlarmList3[2,k1] := 'E38_1.Error Mettler Toledo 2';
			73:
				AlarmList[2,k1] := "E39_1.Lỗi ben chặn sâu đẩy ra trạm 1 [kiểm tra U1I5-7]";
				AlarmList3[2,k1] := 'E39_1.The cylinder blocking worm extend  is faulty line 1';	
			75:
				AlarmList[2,k1] := "E40_1.Lỗi thiếu khí đầu vào [kiểm tra U1I7-13]";
				AlarmList3[2,k1] := 'E40_1.Error of lack of input air [check U1I7-13]';	
			76:
				AlarmList[2,k1] := "E41_1.Lỗi hết thức ăn trạm 1";
				AlarmList3[2,k1] := 'E41_1.Error running out of food line 1';
			77:
				AlarmList[2,k1] := "E42_1.Lỗi hết sâu trạm 1";
				AlarmList3[2,k1] := 'E42_1.Error running out of larvae line 1';		
			98:
				AlarmList[2,k1] := "E98_1.Dừng khẩn [kiểm tra Emergency]";
				AlarmList3[2,k1] := 'E98_1.Emergency Stop [check Emergency]';	 
			99: 
				AlarmList[2,k1] := "E99_1.Lỗi biến tần băng tải đầu ra [kiểm tra biến tần 3]";
				AlarmList3[2,k1] := 'E99_1.The inverter of conveyor out [check inverter 3]';
			101:
				AlarmList[2,k1] := "W1_1.Cảnh báo hết hũ trạm 1[kiểm tra U1I5-2]";
				AlarmList3[2,k1] := 'W1_1.Warning out of jar line 1 [check U1I5-2]';
			102:
				AlarmList[2,k1] := "W2_1.Cảnh báo hết nắp trạm 1[kiểm tra U1I5-8]";
				AlarmList3[2,k1] := 'W2_1.Warning out of lid line 1 [check U1I5-8]';
			103:
				AlarmList[2,k1] := "W3_1.Cảnh báo hết thức ăn trạm 1";
				AlarmList3[2,k1] := 'W3_1.Warning running out of food line 1';
			104:
				AlarmList[2,k1] := "W4_1.Cảnh báo cân quá khối lượng thức ăn trạm 1";
				AlarmList3[2,k1] := 'W4_1.Warning food weight exceeds limit line 1';
			105:
				AlarmList[2,k1] := "W5_1.Cảnh báo hết sâu trạm 1";
				AlarmList3[2,k1] := 'W5_1.Warning running out of larvae line 1';
			106:
				AlarmList[2,k1] := "W6_1.Canh bao can qua khoi luong sau tram 1";
				AlarmList3[2,k1] := 'W6_1.Warning larvae weight exceeds limit line 1';
			107:
				AlarmList[2,k1] := "W7_1.Cảnh báo dập nắp không vô trạm 1[kiểm tra U1I6-7]";
				AlarmList3[2,k1] := 'W7_1.Warning do not press lid inward line 1 [check U1I6-7]';
			115:
				AlarmList[2,k1] := "W8_1.Cảnh báo mất kết nối với PC Advantech [kiểm tra PC]";
				AlarmList3[2,k1] := 'W8_1.Warning disconnect to PC Advantech [check PC]';	
	END_CASE
END_FOR
bWriteAlarm	:= FALSE;
END_IF
END_ACTION

ACTION steError_active:
PR_Line01.Stop();
bStatusStart1 := FALSE;
status := 'ERROR';
bfinish1 := TRUE;
IF i > 100 THEN
	i := 100;
END_IF

CASE nState2 OF 
	0:
		Reset_T(clk := bReset);
		IF Reset_T.Q THEN
			nState2 := 1;
		END_IF
	1:
		timerReset(IN := TRUE, PT := T#500MS);
		PR_Line01.Reset();
		IF nErrorIDList1[1].ErrorStatus = 1 THEN
			IF i <> 1 THEN
				FOR	k := i TO 2 BY -1 DO
				nErrorIDList1[k].nErrorID 	 := nErrorIDList1[k-1].nErrorID;
				nErrorIDList1[k].ErrorTime   := nErrorIDList1[k-1].ErrorTime;
				nErrorIDList1[k].ErrorStatus := nErrorIDList1[k-1].ErrorStatus;		
				END_FOR		
			END_IF 
			nState2 := 2;
		ELSE 
			nState2 := 3;
		END_IF
	2:
		bWriteAlarm	:= TRUE;
		timerReset(IN := TRUE, PT := T#500MS);
		PR_Line01.Reset();
		nErrorIDList1[1].nErrorID := nErrorID;
		nErrorIDList1[1].ErrorTime := SYSTEMTIME_TO_DT(GetLocalSystemTime.systemTime);
		nErrorIDList1[1].ErrorStatus := 0;
		i := i + 1;	
		nState2 := 3;
	3:
		timerReset(IN := TRUE, PT := T#500MS);
		PR_Line01.Reset();
		IF timerReset.Q THEN
			nState2 := 4;
		END_IF
	4:
		timerReset(IN := FALSE);
		Reset_T(clk := FALSE);
		traError := FALSE;
		nState2 := 0;
END_CASE

IF bReset THEN
	bError1 := FALSE;
	bWarning := FALSE;
	bLight_Stop := FALSE;
	bSirens := FALSE;
	status := 'STOP';
	Error[4] := FALSE;
	Error[5] := FALSE;
	Error[7] := FALSE;
	Error[3] := FALSE;
END_IF

IF NOT bEmer THEN
	PR_Line01.Init();
	bRun := FALSE;
END_IF

IF bTo_alarm_side THEN
	VisuElems.CURRENTVISU := 'N_Alarm';
	IF VisuElems.CURRENTVISU = 'N_Alarm' THEN
		bTo_alarm_side := FALSE;
	END_IF
END_IF
END_ACTION

ACTION steErrorCheck_active:

END_ACTION

ACTION steInit_active:
traInitDone := TRUE;
bStatusStart1 := FALSE;
END_ACTION

ACTION steModeAuto_active:
PR_Line01.Auto();
bResetmanual1 := TRUE;
IF bReset THEN
	bWarning := FALSE;
	bSirens  := FALSE;
	bAlarm_Iot := FALSE;
	bWrn 	 := FALSE;
END_IF
END_ACTION

ACTION steModeManual_active:
PR_Line01.Manual();
PR_Line01.Check_reset();
END_ACTION

ACTION steModeSel_active:
IF VisuElems.CURRENTVISU = 'MAIN_LINE1' THEN
	bModeAuto := TRUE;
	bModeManual := FALSE;
END_IF

IF VisuElems.CURRENTVISU = 'N_FoodSupply1' OR VisuElems.CURRENTVISU = 'N_JarSupply1' OR VisuElems.CURRENTVISU = 'N_LidPressing1' OR
	VisuElems.CURRENTVISU = 'N_LidSupply1' OR VisuElems.CURRENTVISU = 'N_Tranfer1' OR VisuElems.CURRENTVISU = 'N_WormWeight1' THEN
	bModeAuto := FALSE;
	bModeManual := TRUE;
END_IF
PR_Line01.check();
bLight_Stop := FALSE;

IF bStart1 THEN
	bStart1 := FALSE;
END_IF
END_ACTION

END_PROGRAM

(* stored: Version 1.1.0.1, ProductVersion 3.1.4024.12
   POU MAIN: Id {888e9e22-ce87-4614-9e28-d2b6f54cee69}, SpecialFunc None
   Folder Mapping: Id {e150aeac-3cf3-4853-b71a-fbb6448f5b7a}
   Action ListError: Id {72a46b4e-20dd-4504-aad3-09ed820a5af3}
   Action MapRtig: Id {c4b49ac0-3b76-48bf-a46e-c8b7f91b0c84}
   Action Reset_active: Id {369709c6-60bc-4c1a-b9f4-f03f517fbd37}
   Action Start_active: Id {b8b28f87-64d5-4713-9744-e7f18a569eff}
   Action steCyclic_active: Id {a9a98539-836f-49c6-8965-f6fd12e74a55}
   Action steError_active: Id {2224a7f2-d2c9-4dcc-a573-f8866e9ca291}
   Action steErrorCheck_active: Id {e300ac53-e6e6-4192-9e29-a77ad1d4b52f}
   Action steInit_active: Id {5601d613-d66f-44f3-8ee5-1391df9c1510}
   Action steModeAuto_active: Id {c0a8b35e-a099-4f25-b577-c61b0c1df42a}
   Action steModeManual_active: Id {9f1d8d52-134c-46ed-ac32-dd59e2feeb0b}
   Action steModeSel_active: Id {47638763-4654-433c-b0e9-e069e1b8d44b} *)
